(* CODESYS project 4 Parking_Garage_counter.project

Project tree, tasks and I/O mapping:
  Device : CODESYS Control Win V3, 3S - Smart Software Solutions GmbH, order no. 305021, version 3.5.7.0
    application Application
      libraries: Standard, * (System)
      task MainTask (cyclic, interval t#20ms, priority 1) calls PLC_PRG
      task VISU_TASK (cyclic, interval 100 ms, priority 31) calls VisuElems.Visu_Prg
      program PLC_PRG [LD]
      visualisation Visualization
  text list GlobalTextList
*)

// Device/Application/PLC_PRG
PROGRAM PLC_PRG
VAR
	start: BOOL;
	stop: BOOL;
	cycle_on: BOOL;
	ext: BOOL;
	entry: BOOL;
	counter_op: BOOL;
	motor: BOOL;
	CTUD_01: CTUD;
	load: BOOL;
	TT: WORD;
END_VAR

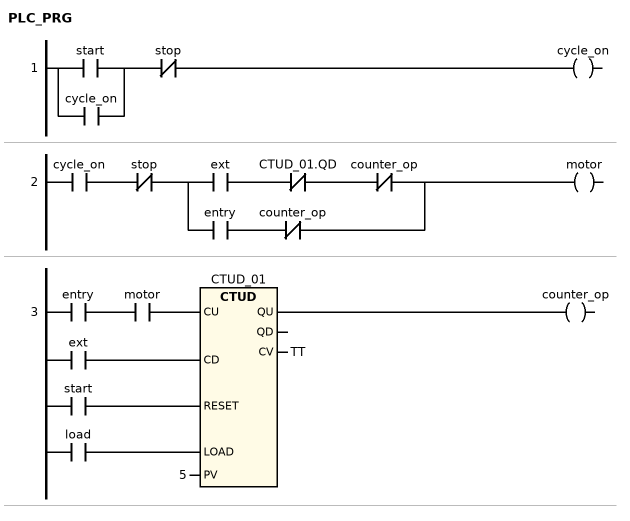
// NETWORK 1
cycle_on := (start OR cycle_on) AND NOT stop;

// NETWORK 2
motor := cycle_on AND NOT stop AND (ext AND NOT CTUD_01.QD AND NOT counter_op OR entry AND NOT counter_op);

// NETWORK 3
CTUD_01(CU := entry AND motor, CD := ext, RESET := start, LOAD := load, PV := 5, CV => TT); // CTUD
counter_op := CTUD_01.QU;

END_PROGRAM

// Device/Application/Visualization
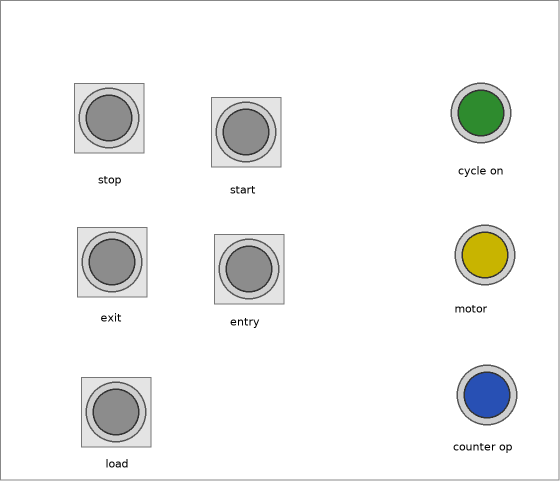
VISUALIZATION Visualization  // 560x481
    PushSwitchLed (74,83 70x70), variable: PLC_PRG.stop, behaviour: TOGGLE, style: Switch-PushSwitchLed-Gray
    PushSwitchLed (211,97 70x70), variable: PLC_PRG.start, behaviour: TOGGLE, style: Switch-PushSwitchLed-Gray
    PushSwitchLed (77,227 70x70), variable: PLC_PRG.ext, behaviour: TOGGLE, style: Switch-PushSwitchLed-Gray
    PushSwitchLed (214,234 70x70), variable: PLC_PRG.entry, behaviour: TOGGLE, style: Switch-PushSwitchLed-Gray
    PushSwitchLed (81,377 70x70), variable: PLC_PRG.load, behaviour: TOGGLE, style: Switch-PushSwitchLed-Gray
    Lamp1 (446,78 70x70), variable: PLC_PRG.cycle_on, style: Lamp-Lamp1-Green
    Lamp1 (450,220 70x70), variable: PLC_PRG.motor, style: Lamp-Lamp1-Yellow
    Lamp1 (452,360 70x70), variable: PLC_PRG.counter_op, style: Lamp-Lamp1-Blue
    Label (35,165 150x30), "stop"
    Label (36,303 150x30), "exit"
    Label (42,449 150x30), "load"
    Label (168,175 150x30), "start"
    Label (170,307 150x30), "entry"
    Label (406,156 150x30), "cycle on"
    Label (396,294 150x30), "motor"
    Label (408,432 150x30), "counter op"
END_VISUALIZATION
